ABB RAPID module: Module1.mod

MODULE Module1
    CONST robtarget pTool1:=[[204.606994476,-1164.704110584,660],[0,-0.258819045,0.965925826,0],[-1,0,-2,0],[9E+09,9E+09,9E+09,9E+09,9E+09,9E+09]];
    CONST robtarget pTool2:=[[-42.943005524,-974.204110584,491.401],[0,-0.707106781,0.707106781,0],[-2,0,-3,0],[9E+09,9E+09,9E+09,9E+09,9E+09,9E+09]];
ENDMODULE
